// TwinCAT 3 PLC project NonInstantFunc
// ProgramVersion: 3.1.4023.0
// libraries:
//   Tc2_Standard, * (Beckhoff Automation GmbH)
//   Tc2_System, * (Beckhoff Automation GmbH)
//   Tc3_Module, * (Beckhoff Automation GmbH)
// project tree:
//   / PlcTask.TcTTO
//   POUs/ CheckFault.TcPOU, MAIN.TcPOU, Prg_NonInstantFunc.TcPOU
// real-time tasks:
//   TASK PlcTask: cycle T#10ms, priority 20, ADS port 350

CONFIGURATION NonInstantFunc
    RESOURCE PLC ON TwinCAT3
        TASK PlcTask(INTERVAL := T#10ms, PRIORITY := 20);
        PROGRAM MAIN WITH PlcTask : MAIN;
    END_RESOURCE
END_CONFIGURATION

// ---- POUs/MAIN.TcPOU
PROGRAM MAIN
VAR
END_VAR

Prg_NonInstantFunc();

END_PROGRAM

// ---- POUs/Prg_NonInstantFunc.TcPOU
PROGRAM Prg_NonInstantFunc
VAR
	Buttons: ARRAY[1..4] OF BOOL;
	Temp: ARRAY[1..4] OF INT := [90, 20, 100, 75];
	OverLoad: ARRAY[1..4] OF BOOL;
	AnalogSensor: ARRAY[1..4] OF INT := [8, 0, 8, 0];
	Coils: ARRAY[1..4] OF BOOL;
	
	i: INT;
	
END_VAR

FOR i:=1 TO 4 BY 1 DO
	IF CheckFault(Overload:=OverLoad[i], MotorTemp:=Temp[i]) THEN
		Coils[i]:=FALSE;
	ELSIF Buttons[i] THEN
		Coils[i]:=TRUE;
	ELSE
		Coils[i]:=FALSE;		
	END_IF
END_FOR

END_PROGRAM

// ---- POUs/CheckFault.TcPOU
FUNCTION CheckFault : BOOL
VAR_INPUT
	Overload: BOOL;
	MotorTemp: INT;
	
END_VAR
VAR
END_VAR

IF Overload OR MotorTemp > 80 THEN
	CheckFault:=TRUE;
ELSE
	CheckFault:=FALSE;
END_IF

END_FUNCTION
